// TwinCAT 3 PLC project SirupAutomat
// ProgramVersion: 3.1.0.5
// libraries:
//   Tc2_Standard, * (Beckhoff Automation GmbH)
//   Tc2_System, * (Beckhoff Automation GmbH)
//   Tc3_Interfaces, * (Beckhoff Automation GmbH)
//   Tc3_Module, * (Beckhoff Automation GmbH)
//   Tc2_OpcUa,3.3.2.0,Beckhoff Automation GmbH
//   Tc2_TcpIp,3.3.1.0,Beckhoff Automation GmbH
//   Tc2_Utilities,3.3.5.0,Beckhoff Automation GmbH
// project tree:
//   DUTs/ EKey.TcDUT, EMethod.TcDUT, EStatus.TcDUT, ECommand.TcDUT, EDosingState.TcDUT, ETimerState.TcDUT, ST_ApplicationBinaryData.TcDUT, ST_BinaryFrame.TcDUT, ST_BinaryHeader.TcDUT
//   GVLs/ DosingOuput.TcGVL, Global_Variables.TcGVL, IOStates.TcGVL, Liquids.TcGVL
//   / I_DigitalOut.TcIO, I_DosingStation.TcIO, PlcTask.TcTTO, Visualization Manager.TcVMO (not stored)
//   POUs/ FB_HardStuffDosingStation.TcPOU, FB_CO2_DosingStation.TcPOU, FB_LocalServer.TcPOU, FB_Timer.TcPOU, FB_DigitalOut.TcPOU, MAIN.TcPOU, FB_DosingStation.TcPOU
//   POUs/IP_POUs/ FB_FrameBinaryFifo.TcPOU, FB_ProtErrorFifo.TcPOU, FB_ServerApplication.TcPOU, F_ADSLOGERROR.TcPOU, F_ADSLOGHEXDATA.TcPOU, SCODE_CODE.TcPOU
//   VISUs/ HardStuff.TcVIS
// real-time tasks:
//   TASK PlcTask: cycle T#1ms, priority 20, ADS port 350
// I/O:
//   DEVICE Device 1 (EtherCAT), AmsNetId 192.168.0.103.2.1
//     Term 6 (EK1200) [EK1200-5000 EtherCAT Power supply (2A E-Bus)]
//       Term 7 (EL1008) [EL1008 8Ch. Dig. Input 24V, 3ms]
//       Term 8 (EL2008) [EL2008 8Ch. Dig. Output 24V, 0.5A]
//       Term 9 (EL2008) [EL2008 8Ch. Dig. Output 24V, 0.5A]
//       Term 10 (EL3061) [EL3061 1Ch. Ana. Input 0-10V]
//       Term 11 (EL9011) [EL9011 End Terminal]
// variable links:
//   SirupAutomat/SirupAutomat Instance <-> Device 1 (EtherCAT)/Term 6 (EK1200)/Term 10 (EL3061)
//     PlcTask Inputs/DosingOuput.iPressure <-> AI Standard/Value
//   SirupAutomat/SirupAutomat Instance <-> Device 1 (EtherCAT)/Term 6 (EK1200)/Term 7 (EL1008)
//     PlcTask Inputs/MAIN.bManualStart <-> Channel 8/Input
//     PlcTask Inputs/MAIN.fbDosingStation1.bPrefill <-> Channel 1/Input
//     PlcTask Inputs/MAIN.fbDosingStation2.bPrefill <-> Channel 2/Input
//     PlcTask Inputs/MAIN.fbDosingStation3.bPrefill <-> Channel 3/Input
//     PlcTask Inputs/MAIN.bGlassPresent <-> Channel 7/Input
//   SirupAutomat/SirupAutomat Instance <-> Device 1 (EtherCAT)/Term 6 (EK1200)/Term 8 (EL2008)
//     PlcTask Outputs/MAIN.fbDosingStation1.fbValve2.bOutput <-> Channel 2/Output
//     PlcTask Outputs/MAIN.fbDosingStation3.fbValve2.bOutput <-> Channel 6/Output
//     PlcTask Outputs/MAIN.fbDosingStation2.fbValve2.bOutput <-> Channel 4/Output
//     PlcTask Outputs/MAIN.fbDosingStation3.fbValve1.bOutput <-> Channel 5/Output
//     PlcTask Outputs/MAIN.fbDosingStation2.fbValve1.bOutput <-> Channel 3/Output
//     PlcTask Outputs/MAIN.fbDosingStation1.fbValve1.bOutput <-> Channel 1/Output
//   SirupAutomat/SirupAutomat Instance <-> Device 1 (EtherCAT)/Term 6 (EK1200)/Term 9 (EL2008)
//     PlcTask Outputs/DosingOuput.bBlowOff <-> Channel 8/Output
//     PlcTask Outputs/DosingOuput.bPump <-> Channel 7/Output

CONFIGURATION SirupAutomat
    RESOURCE PLC ON TwinCAT3
        TASK PlcTask(INTERVAL := T#1ms, PRIORITY := 20);
        PROGRAM MAIN WITH PlcTask : MAIN;
    END_RESOURCE
END_CONFIGURATION

// ---- DUTs/EKey.TcDUT
TYPE EKey :
(
	KeyCommand := 1,
	KeyVolume := 2,
	KeyStationID := 3,
	KeyStatus := 4
);
END_TYPE

// ---- DUTs/EMethod.TcDUT
TYPE EMethod :
(
	MethGet := 1,
	MethPut := 2,
	MethResponse := 3
);
END_TYPE

// ---- DUTs/EStatus.TcDUT
TYPE EStatus :
(
	NotReady,
	Ready,
	Prefilling,
	DeliverLiquid,
	Error,
	PreparingForNextDrink,
	MeasuringContent,
	RunningManualDeliver
);
END_TYPE

// ---- DUTs/ECommand.TcDUT
TYPE ECommand :
(
	None := 0,
	Deliver := 1,
	ErrorAck := 2,
	PrepareForNextDrink := 3,
	MeasureContent := 4,
	StartManualCycle
);
END_TYPE

// ---- DUTs/EDosingState.TcDUT
TYPE EDosingState :
(
	eStopped,
	eV1Opened,
    eV1AndV3Opened,
	eV1AndV2AndV3Closed,
	eV2Opened,
    eV3Opened,
	eP1Started,
	eP1Stopped,
	eV1Stopped,
	eEnd
);
END_TYPE

// ---- DUTs/ETimerState.TcDUT
TYPE ETimerState :
(
	created := 0,
	started := 1,
	outputHigh := 2,
	outputLow := 3
);
END_TYPE

// ---- DUTs/ST_ApplicationBinaryData.TcDUT
TYPE ST_ApplicationBinaryData :(* Example of binary user data structure (4 byte aligned) *)
STRUCT
	(* Adapt this structure to match your protocol needs *)
	dwMethode : DWORD;
	dwKey : DWORD;
	dwValue : DWORD;
	(* total user data size = 120 byte *)
END_STRUCT
END_TYPE

// ---- DUTs/ST_BinaryFrame.TcDUT
TYPE ST_BinaryFrame :(* Simple binary TCP/IP frame (4 byte aligned) *)
STRUCT
	head	:  ST_BinaryHeader;(* frame header *)
	data 	: ARRAY[1..PLCPRJ_BUFFER_SIZE] OF BYTE; (* user data of max. length *)
END_STRUCT
END_TYPE

// ---- DUTs/ST_BinaryHeader.TcDUT
TYPE ST_BinaryHeader :(* Simple frame header (4 byte aligned) *)
STRUCT
	dwHead		: DWORD	:= 16#BECF1234;	(* start bytes *)
	cbLength		: UDINT(0..PLCPRJ_BUFFER_SIZE) := 0;(* Max. length of attached binary data *)
	nS			: UDINT 		:= 0;		(* send counter *)
	nR			: UDINT		:= 0;		(* receive counter *)
END_STRUCT
END_TYPE

// ---- GVLs/DosingOuput.TcGVL
VAR_GLOBAL
    bPump AT %Q* : BOOL;
    bBlowOff AT %Q* : BOOL;
	iPressure AT %I* : INT;
END_VAR

// ---- GVLs/Global_Variables.TcGVL
VAR_GLOBAL CONSTANT
	PLCPRJ_MAX_CONNECTIONS						: UDINT 	:= 5;(* Max. number of server<->client connections *)
	PLCPRJ_SERVER_RESPONSE_TIMEOUT			: TIME 	:= T#10s;
	PLCPRJ_CLIENT_SEND_CYCLE_TIME				: TIME 	:= T#1s;

	PLCPRJ_RECEIVER_POLLING_CYCLE_TIME			: TIME 	:= T#200ms;
	PLCPRJ_BUFFER_SIZE							: UDINT 	:= 10000;(* Max. internal fifo/receiver buffer size *)

	(* Some project specific error codes *)
	PLCPRJ_ERROR_RECEIVE_BUFFER_OVERFLOW	: UDINT := 16#8101; (* receive fifo/buffer overflow*)
	PLCPRJ_ERROR_SEND_BUFFER_OVERFLOW		: UDINT := 16#8102;(* send fifo/buffer overflow *)
	PLCPRJ_ERROR_RESPONSE_TIMEOUT			: UDINT := 16#8103;(* receive timeout error *)
	PLCPRJ_ERROR_INVALID_FRAME_FORMAT		: UDINT := 16#8104;(* invalid frame format/data *)
END_VAR

// ---- GVLs/IOStates.TcGVL
VAR_GLOBAL
	byteInletValves AT %QB1 : BYTE;
END_VAR

// ---- GVLs/Liquids.TcGVL
VAR_GLOBAL
	Status AT %Q* : EStatus := NotReady; (*~	(OPC : 1 : available for OPC-clients)	*)
	Command AT %I* : ECommand := None; (*~	(OPC : 1 : available for OPC-clients)	*)
	StationID  AT %I* : UINT := 0; (*~	(OPC : 1 : available for OPC-clients)	*)
	Volume_ml  AT %I* : UINT := 0; (*~	(OPC : 1 : available for OPC-clients)	*)
	ErrString  AT %Q* : STRING := ''; (*~	(OPC : 1 : available for OPC-clients)	*)
	GlassPresent : BOOL := FALSE;
END_VAR

// ---- I_DigitalOut.TcIO
INTERFACE I_DigitalOut

METHOD M_On
VAR_INPUT
END_VAR
END_METHOD

 METHOD M_Off
VAR_INPUT
END_VAR
END_METHOD

END_INTERFACE

// ---- I_DosingStation.TcIO
INTERFACE I_DosingStation

METHOD M_Fill
VAR_INPUT
	tiPumpTime : TIME;
END_VAR
END_METHOD

METHOD M_Prefill
VAR_INPUT
END_VAR
END_METHOD

METHOD M_Stop
VAR_INPUT
END_VAR
END_METHOD

METHOD M_PrepareForNextDrink
VAR_INPUT
END_VAR
END_METHOD

METHOD M_GetContent_ml : BOOL
VAR_INPUT
END_VAR
END_METHOD

END_INTERFACE

// ---- POUs/MAIN.TcPOU
PROGRAM MAIN
VAR
	iStationIndex : UINT := 0;
	bGlassPresent AT %I* : BOOL;
	bManualStart AT %I* : BOOL;
	// systemState : ESystemState := eStandby;
    
	fbDosingStation1 : FB_HardStuffDosingStation;
	fbDosingStation2 : FB_HardStuffDosingStation;
    fbDosingStation3 : FB_CO2_DosingStation;
	DeliveryLiquid: INT;
	duration : TIME;
	
	A_Prefilling: INT;
	
	sLocalHost	: STRING(15) 	:= '0.0.0.0';(* Server address *)
	nLocalPort	: UDINT 		:= 200;(* Server port number *)
	bEnable		: BOOL 		:= TRUE;(* TRUE => enable server data exchange, FALSE => disable *)
	hServer		: T_HSERVER;(* Server connection handle *)
	fbApplication	: FB_ServerApplication := ( bDbg:=FALSE );(* Application (connection) instances *)

	fbCloseAll	: FB_SocketCloseAll;
	bCloseAll	: BOOL := TRUE;
	
END_VAR

A_RunIP();

CASE Status OF
	NotReady :
		IF bGlassPresent = TRUE THEN
			Status := Ready;
		ELSE
			// this works only, when no glass is present
			IF Command = MeasureContent THEN
				Status := MeasuringContent;
				iStationIndex := StationID;
				Command := None;
			END_IF
		END_IF
		
	Ready:
		IF bGlassPresent = FALSE THEN
			Status := NotReady;  
		END_IF
		
		IF Command = Deliver THEN
			Status := DeliverLiquid;
			Command := None;
		ELSIF Command = PrepareForNextDrink THEN
			Status := PreparingForNextDrink;
			Command := None;
		ELSE
			IF fbDosingStation1.bPrefill THEN 
				iStationIndex := 1;
				Status := Prefilling;
			ELSIF fbDosingStation2.bPrefill THEN
				iStationIndex := 2;
				Status := Prefilling;
			ELSIF fbDosingStation3.bPrefill THEN
				iStationIndex := 3;
				Status := Prefilling;
			ELSIF bManualStart THEN
				iStationIndex := 0;
				Status := RunningManualDeliver;
			END_IF	
		END_IF
	MeasuringContent:
		A_MeasureContent();
  
	Prefilling:
		A_Prefill();
		
	RunningManualDeliver:
		A_MixACubaLibre();
	
	DeliverLiquid:
		duration := INT_TO_TIME(UINT_TO_INT(Volume_ml) * 111);
		CASE StationID OF
			1:
				IF bGlassPresent = FALSE THEN
					fbDosingStation1.M_Stop();
					Status := Error;
				ELSE
					fbDosingStation1.M_Fill(duration);
					IF fbDosingStation1.bFinished THEN
						Status := NotReady;
					END_IF
				END_IF
		
			2:
				IF bGlassPresent = FALSE THEN
					fbDosingStation2.M_Stop();
					Status := Error;
				ELSE
					fbDosingStation2.M_Fill(duration);
					IF fbDosingStation2.bFinished THEN
						Status := NotReady;
					END_IF
				END_IF
				
			3:
				IF bGlassPresent = FALSE THEN
					fbDosingStation3.M_Stop();
					Status := Error;
				ELSE
					fbDosingStation3.M_Fill(duration);
					IF fbDosingStation3.bFinished THEN
						Status := NotReady;
					END_IF
				END_IF		
	
		END_CASE

	Error:
		IF Command = ErrorAck THEN
			Status := NotReady;
		END_IF
		
	PreparingForNextDrink:
		CASE StationID OF
			1:
				IF bGlassPresent = FALSE THEN
					fbDosingStation1.M_Stop();
					Status := Error;
				ELSE
					fbDosingStation1.M_PrepareForNextDrink();
					IF fbDosingStation1.bFinished THEN
						Status := NotReady;
					END_IF
				END_IF
		
			2:
				IF bGlassPresent = FALSE THEN
					fbDosingStation2.M_Stop();
					Status := Error;
				ELSE
					fbDosingStation2.M_PrepareForNextDrink();
					IF fbDosingStation2.bFinished THEN
						Status := NotReady;
					END_IF
				END_IF
				
			3:
				IF bGlassPresent = FALSE THEN
					fbDosingStation3.M_Stop();
					Status := Error;
				ELSE
					fbDosingStation3.M_PrepareForNextDrink();
					IF fbDosingStation3.bFinished THEN
						Status := NotReady;
					END_IF
				END_IF		
	
		END_CASE		
		
END_CASE

ACTION A_Prefill:
IF iStationIndex = 1 THEN
    fbDosingStation1.M_Prefill();
    IF fbDosingStation1.bFinished THEN
		iStationIndex := 0;
		Status := NotReady;
    END_IF
ELSIF  iStationIndex = 2  THEN
    fbDosingStation2.M_Prefill();
    IF fbDosingStation2.bFinished THEN
		iStationIndex := 0;
		Status := NotReady;
    END_IF
ELSIF  iStationIndex = 3  THEN
    fbDosingStation3.M_Prefill();
    IF fbDosingStation3.bFinished THEN
		iStationIndex := 0;
		Status := NotReady;
    END_IF
END_IF
END_ACTION

ACTION A_RunIP:
IF bCloseAll THEN(*On PLC reset or program download close all old (opened) connections *)
	bCloseAll := FALSE;

	(* Initialize server handle *)
	F_CreateServerHnd( 	sSrvNetID 	:= '',
						sLocalHost 	:= sLocalHost,
						nLocalPort	:= nLocalPort,
						nMode 		:= CONNECT_MODE_ENABLEDBG,(* Enable debug messages *)
						bEnable 		:= FALSE,(* TRUE = leave listener socket open, FALSE = close listener socket after last connection ist closed too *)
						hServer 		:= hServer );


	fbCloseAll( bExecute:= TRUE );
ELSE
	fbCloseAll( bExecute:= FALSE );
END_IF


IF NOT fbCloseAll.bBusy THEN
	(* trigger the execution of every connection instance *)
	fbApplication( hServer := hServer, bEnable := bEnable );
END_IF
END_ACTION

ACTION A_MeasureContent:
IF iStationIndex = 1 THEN
    fbDosingStation1.M_GetContent_ml();
    IF fbDosingStation1.bFinished THEN
		iStationIndex := 0;
		Status := NotReady;
    END_IF
ELSIF  iStationIndex = 2  THEN
    fbDosingStation2.M_GetContent_ml();
    IF fbDosingStation2.bFinished THEN
		iStationIndex := 0;
		Status := NotReady;
    END_IF
ELSIF  iStationIndex = 3  THEN
    fbDosingStation3.M_GetContent_ml();
    IF fbDosingStation3.bFinished THEN
		iStationIndex := 0;
		Status := NotReady;
    END_IF
END_IF
END_ACTION

ACTION A_MixACubaLibre:
IF iStationIndex = 0 THEN
    iStationIndex := 3;
END_IF

IF iStationIndex = 1 THEN
    // the Rum
	fbDosingStation1.M_Fill(INT_TO_TIME(UINT_TO_INT(10) * 111));
    IF fbDosingStation1.bFinished THEN
        iStationIndex := 4;
    END_IF
END_IF

IF iStationIndex = 2 THEN
    // the Vodka is not used yet 
	fbDosingStation2.M_Fill(TIME#16S);
    IF fbDosingStation2.bFinished THEN
        iStationIndex := 3;
    END_IF
END_IF

IF iStationIndex = 3 THEN
    // the CocaCola 
	fbDosingStation3.M_Fill(INT_TO_TIME(UINT_TO_INT(200) * 111));
    IF fbDosingStation3.bFinished THEN
        iStationIndex := 1;
    END_IF
END_IF

IF iStationIndex = 4 THEN
    iStationIndex := 0;
	Status := NotReady;
END_IF
END_ACTION

END_PROGRAM

// ---- POUs/FB_HardStuffDosingStation.TcPOU
FUNCTION_BLOCK FB_HardStuffDosingStation EXTENDS FB_DosingStation
VAR_INPUT
	bPrefill AT %I* : BOOL;
END_VAR
VAR_OUTPUT
	bFinished : BOOL := TRUE;
	error : BOOL := FALSE;
END_VAR
VAR
	fbT1 : FB_Timer;
	dosingState : EDosingState := eStopped;
	fbValve1 : FB_DigitalOut;
	fbValve2 : FB_DigitalOut;
	
	iStartPressure : INT;
	iActualPressure : INT;
	iDeltaPressure : INT;
	iContentMeasurementTimeout : TIME := TIME#5S;
END_VAR
VAR_EXTERNAL
    bPump : BOOL;
END_VAR

;

METHOD M_Fill
VAR_INPUT
	    tiPumpTime : TIME := TIME#2S;
END_VAR

CASE dosingState OF
	eStopped :
		// wait for start
   		bFinished := FALSE;
        fbValve2.M_On();
        dosingState := eV2Opened;
	eV2Opened :
		fbT1.M_Start(TIME#1S);
		IF fbT1.bTimeout THEN
			fbValve1.M_On();
			dosingState := eV1Opened;
		END_IF
	eV1Opened :
		fbT1.M_Start(TIME#1S);
		IF fbT1.bTimeout THEN
			bPump := TRUE;
			dosingState := eP1Started;
		END_IF
	eP1Started :
		fbT1.M_Start(tiPumpTime);
		IF fbT1.bTimeout THEN
			bPump := FALSE;
			dosingState := eP1Stopped;
		END_IF
	eP1Stopped :
		fbT1.M_Start(TIME#1S);
		IF fbT1.bTimeout THEN
			fbValve1.M_Off();
			dosingState := eV1Stopped;
		END_IF
	eV1Stopped :
		fbT1.M_Start(TIME#10S);
		IF fbT1.bTimeout THEN
			fbValve2.M_Off();
			dosingState := eEnd;
		END_IF
	eEnd :
   		bFinished := TRUE;
		dosingState := eStopped;
END_CASE
END_METHOD

METHOD M_Prefill
VAR_INPUT
END_VAR
CASE dosingState OF
	eStopped :
		// wait for start
   		bFinished := FALSE;
        fbValve2.M_On();
        dosingState := eV2Opened;
	eV2Opened :
		fbT1.M_Start(TIME#0S);
		IF fbT1.bTimeout THEN
			fbValve1.M_On();
			dosingState := eV1Opened;
		END_IF
	eV1Opened :
		fbT1.M_Start(TIME#0S);
		IF fbT1.bTimeout THEN
			bPump := TRUE;
			dosingState := eP1Started;
		END_IF
	eP1Started :
		IF NOT bPrefill THEN
			bPump := FALSE;
			dosingState := eP1Stopped;
		END_IF
	eP1Stopped :
		fbT1.M_Start(TIME#1S);
		IF fbT1.bTimeout THEN
			fbValve1.M_Off();
			dosingState := eV1Stopped;
		END_IF
	eV1Stopped :
		fbT1.M_Start(TIME#5S);
		IF fbT1.bTimeout THEN
			fbValve2.M_Off();
			dosingState := eEnd;
		END_IF
	eEnd :
   		bFinished := TRUE;
		dosingState := eStopped;
END_CASE
END_METHOD

METHOD M_Stop
VAR_INPUT
END_VAR
fbValve2.M_Off();
fbValve1.M_Off();
bPump := FALSE;	
dosingState := eStopped;
bFinished := TRUE;
END_METHOD

METHOD M_PrepareForNextDrink
VAR_INPUT
END_VAR
CASE dosingState OF
	eStopped :
		// wait for start
		bFinished := FALSE;
        fbValve2.M_On();
        dosingState := eV2Opened;
	eV2Opened :
		fbT1.M_Start(TIME#10S);
		IF fbT1.bTimeout THEN
			fbValve2.M_Off();
			dosingState := eEnd;
		END_IF
	eEnd :
   		bFinished := TRUE;
		dosingState := eStopped;		
END_CASE
END_METHOD

METHOD M_GetContent_ml : BOOL
VAR_INPUT
END_VAR
VAR
END_VAR
CASE dosingState OF
	eStopped :
		// wait for start
   		bFinished := FALSE;
        // open the 2 valves (the blow off valve is valve 3) to release overpressure of the CO2 bottle
        bBlowOff := TRUE;
        fbValve1.M_On();
        dosingState := eV1AndV3Opened;
    eV1AndV3Opened :    
		fbT1.M_Start(TIME#2S);
		IF fbT1.bTimeout THEN
            // after a timeout close the blow off valve and the inlet
			bBlowOff := FALSE;
			fbValve1.M_Off();
			iStartPressure := iPressure;
			bPump := TRUE;
			dosingState := eV1AndV2AndV3Closed;
		END_IF
	eV1AndV2AndV3Closed :
		// now everything is closed, pump it up
		fbT1.M_Start(iContentMeasurementTimeout);
		IF fbT1.bTimeout THEN
			iActualPressure := iPressure;
			bPump := FALSE;
			// let the pressure escape
			bBlowOff := TRUE;
			dosingState := eV3Opened;
		END_IF
	eV3Opened :
		fbT1.M_Start(TIME#1S);
		IF fbT1.bTimeout THEN
			iDeltaPressure := iActualPressure - iStartPressure;
			bBlowOff := FALSE;
			dosingState := eEnd;
		END_IF
	eEnd :
   		bFinished := TRUE;
		dosingState := eStopped;
END_CASE
END_METHOD

END_FUNCTION_BLOCK

// ---- POUs/FB_DosingStation.TcPOU
FUNCTION_BLOCK FB_DosingStation IMPLEMENTS I_DosingStation
VAR_INPUT
END_VAR
VAR_OUTPUT
END_VAR
VAR
END_VAR

METHOD M_Fill
VAR_INPUT
	tiPumpTime : TIME;
END_VAR
END_METHOD

METHOD M_Prefill
VAR_INPUT
END_VAR
END_METHOD

METHOD M_Stop
VAR_INPUT
END_VAR
END_METHOD

METHOD M_PrepareForNextDrink
VAR_INPUT
END_VAR
END_METHOD

METHOD M_GetContent_ml : BOOL
VAR_INPUT
END_VAR
;
END_METHOD

END_FUNCTION_BLOCK

// ---- POUs/FB_Timer.TcPOU
FUNCTION_BLOCK FB_Timer
VAR_INPUT
	tiTimeout : TIME;
END_VAR
VAR_OUTPUT
	bTimeout : BOOL;
	iIndex : UINT := 0;
	toggler : BOOL := FALSE;
END_VAR
VAR
	timer : TON;
	toggleTimer : TON;
	countUpTimer : TON;
	elapsed : TIME;
	state : ETimerState := created;
END_VAR

;

METHOD M_ToggleOutput
VAR_INPUT
END_VAR
elapsed := toggleTimer.ET;
CASE state OF 
	created :
		//onTimer.PT := TIME#4S;
		toggleTimer(IN := TRUE, PT := TIME#4S);
		state := outputLow;
	outputLow :
		IF NOT toggleTimer.Q THEN
			toggleTimer(IN := TRUE, PT := TIME#1S);
		END_IF
		IF toggleTimer.Q THEN
			toggleTimer(IN := FALSE);
			state := outputHigh;
			toggler := TRUE;
		END_IF
	outputHigh :		
		IF NOT toggleTimer.Q THEN
			toggleTimer(IN := TRUE, PT := TIME#1S);
		END_IF
		IF toggleTimer.Q THEN
			toggleTimer(IN := FALSE);
			state := outputLow;
			toggler := FALSE;
		END_IF
END_CASE
END_METHOD

METHOD M_CountUp
VAR_INPUT
END_VAR
IF NOT countUpTimer.Q THEN
	countUpTimer( IN := TRUE, PT := TIME#2S );
END_IF

IF countUpTimer.Q THEN
	countUpTimer( IN := FALSE ); 
	iIndex := iIndex + 1;
END_IF
END_METHOD

METHOD M_Start
VAR_INPUT
	tiTimeout : TIME;
END_VAR
IF NOT timer.Q THEN
	bTimeout := FALSE; 
	timer( IN := TRUE, PT := tiTimeout );
END_IF

IF timer.Q THEN
	timer( IN := FALSE );
	bTimeout := TRUE; 
END_IF
timer();
END_METHOD

END_FUNCTION_BLOCK

// ---- POUs/FB_DigitalOut.TcPOU
FUNCTION_BLOCK FB_DigitalOut IMPLEMENTS I_DigitalOut
VAR_INPUT
END_VAR
VAR_OUTPUT
	bOutput AT %Q* : BOOL := FALSE;
END_VAR
VAR
END_VAR

METHOD M_Off
bOutput := FALSE;
END_METHOD

METHOD M_On
bOutput := TRUE;
END_METHOD

END_FUNCTION_BLOCK

// ---- POUs/FB_CO2_DosingStation.TcPOU
FUNCTION_BLOCK FB_CO2_DosingStation  IMPLEMENTS I_DosingStation
VAR_INPUT
	bPrefill AT %I* : BOOL;
END_VAR
VAR_OUTPUT
	bFinished : BOOL := TRUE;
END_VAR
VAR
	fbT1 : FB_Timer;
	dosingState : EDosingState := eStopped;
	fbValve1 : FB_DigitalOut;
	fbValve2 : FB_DigitalOut;
END_VAR
VAR_EXTERNAL
    // the global enable/disable for the pump and the blow off valve
    bPump : BOOL;
    bBlowOff : BOOL;
END_VAR

;

METHOD M_Fill
VAR_INPUT
    tiPumpTime : TIME := TIME#2S;
END_VAR
CASE dosingState OF
	eStopped :
		// wait for start
   		bFinished := FALSE;
        // open the 2 valves (the blow off valve is valve 3) to release overpressure of the CO2 bottle
        bBlowOff := TRUE;
        fbValve1.M_On();
        dosingState := eV1AndV3Opened;
    eV1AndV3Opened :    
		fbT1.M_Start(TIME#2S);
		IF fbT1.bTimeout THEN
            // after a timeout close the blow off valve and open the outlet
			bBlowOff := FALSE;
			fbValve2.M_On();
			dosingState := eV2Opened;
		END_IF
	eV2Opened :
		fbT1.M_Start(TIME#1S);
		IF fbT1.bTimeout THEN
			fbValve1.M_On();
			dosingState := eV1Opened;
		END_IF
	eV1Opened :
		fbT1.M_Start(TIME#1S);
		IF fbT1.bTimeout THEN
			bPump := TRUE;
			dosingState := eP1Started;
		END_IF
	eP1Started :
		fbT1.M_Start(tiPumpTime);
		IF fbT1.bTimeout THEN
			bPump := FALSE;
			dosingState := eP1Stopped;
		END_IF
	eP1Stopped :
		fbT1.M_Start(TIME#1S);
		IF fbT1.bTimeout THEN
			fbValve1.M_Off();
			dosingState := eV1Stopped;
		END_IF
	eV1Stopped :
		fbT1.M_Start(TIME#10S);
		IF fbT1.bTimeout THEN
			fbValve2.M_Off();
			dosingState := eEnd;
		END_IF
	eEnd :
   		bFinished := TRUE;
		dosingState := eStopped;
END_CASE
END_METHOD

METHOD M_Prefill
VAR_INPUT
END_VAR
CASE dosingState OF
	eStopped :
		// wait for start
		bFinished := FALSE;
		// open the 2 valves (the blow-off valve an inlet of the bottle) to release overpressure of the CO2 bottle
		bBlowOff := TRUE;
		fbValve1.M_On();
		dosingState := eV1AndV3Opened;
	eV1AndV3Opened :
        // let the CO2 blow-off for a short time    
		fbT1.M_Start(TIME#2S);
		IF fbT1.bTimeout THEN
			// after a timeout close the blow-off valve and open the outlet
            // let the inlet open
			bBlowOff := FALSE;
			fbValve2.M_On();
            // jump directly to the pump, because the inlet ist already open
			dosingState := eV1Opened;
		END_IF
	eV2Opened :
        // don't wait 
		fbT1.M_Start(TIME#0S);
		IF fbT1.bTimeout THEN
			fbValve1.M_On();
			dosingState := eV1Opened;
		END_IF
	eV1Opened :
        // don't wait 
		fbT1.M_Start(TIME#0S);
		IF fbT1.bTimeout THEN
			bPump := TRUE;
			dosingState := eP1Started;
		END_IF
	eP1Started :
		IF NOT bPrefill THEN
			bPump := FALSE;
			dosingState := eP1Stopped;
		END_IF
	eP1Stopped :
        // don't wait the Coca Cola pooring out
        // therefore close inlet and outlet simultaneously
		fbT1.M_Start(TIME#0S);
		IF fbT1.bTimeout THEN
			fbValve1.M_Off();
			fbValve2.M_Off();
			dosingState := eEnd;
		END_IF
	eV1Stopped :
		fbT1.M_Start(TIME#5S);
		IF fbT1.bTimeout THEN
			fbValve2.M_Off();
			dosingState := eEnd;
		END_IF
	eEnd :
		bFinished := TRUE;
		dosingState := eStopped;
END_CASE
END_METHOD

METHOD M_Stop
VAR_INPUT
END_VAR
fbValve2.M_Off();
fbValve1.M_Off();
bPump := FALSE;	
dosingState := eStopped;
bFinished := TRUE;
END_METHOD

METHOD M_PrepareForNextDrink
VAR_INPUT
END_VAR
bFinished := TRUE;
dosingState := eStopped;
END_METHOD

METHOD M_GetContent_ml : BOOL
VAR_INPUT
END_VAR
VAR
	uiStartPressure : UINT;
	uiActualPressure : UINT;
END_VAR
;
END_METHOD

END_FUNCTION_BLOCK

// ---- POUs/IP_POUs/FB_ServerApplication.TcPOU
FUNCTION_BLOCK FB_ServerApplication
(* Sample server application. Adapt this code to match your needs. *)
VAR_IN_OUT
	hServer 	: T_HSERVER;(* Server connection handle *)
END_VAR
VAR_INPUT
	bDbg		: BOOL 	:= FALSE;(* TRUE => Enable debug output, FALSE => Disable *)
	bEnable		: BOOL 	:= TRUE;(* TRUE => Enable connection, FALSE => Disable *)
END_VAR
VAR_OUTPUT
	eState		: E_SocketConnectionState := eSOCKET_DISCONNECTED;(* TCP/IP connection state *)
END_VAR
VAR
	bCaseError : BOOL;
	fromClient	: ST_ApplicationBinaryData; (* Rx user data *)
	toClient	: ST_ApplicationBinaryData; (* Tx user data *)

	fbServer		: FB_LocalServer;(* Implements one server->client connection *)
	tx 			: FB_FrameBinaryFifo; (* Tx fifo *)
	rx 			: FB_FrameBinaryFifo; (* Rx fifo *)
	errors		: FB_ProtErrorFifo; (* Error fifo *)
END_VAR

(* ------------------------------------- trigger data exchange ----------------------------------------------------------------------------------------------*)
fbServer( bDbg := bDbg, hServer := hServer, rx := rx, tx := tx, errors := errors, bEnable := bEnable, eState => eState  );



(*----------------------------------------------- fetch rx data and send them back to the client ---------------------------------------------------------------------------------------------------- *)
IF eState = eSOCKET_CONNECTED THEN

	REPEAT
		rx.A_RemoveHead( pGet := ADR( fromClient ), cbGet := SIZEOF( fromClient ) );(* fetch data from rx fifo *)
		IF rx.bOk THEN(* success *)

			IF fromClient.dwMethode = MethPut THEN
				CASE fromClient.dwKey OF
					KeyCommand:
						Command  := DWORD_TO_INT(fromClient.dwValue);
						bCaseError := FALSE;
					KeyVolume:
						Volume_ml := DWORD_TO_INT(fromClient.dwValue);
						bCaseError := FALSE;
					KeyStationID:
					    StationID := DWORD_TO_INT(fromClient.dwValue);
						bCaseError := FALSE;
				ELSE
					bCaseError := TRUE;
				END_CASE
				// don't leave him with no response
				toClient.dwMethode := MethResponse;
				toClient.dwKey := fromClient.dwKey;
				toClient.dwValue := fromClient.dwValue;
			ELSIF  fromClient.dwMethode = MethGet THEN
				CASE fromClient.dwKey OF
					KeyStatus:
						toClient.dwMethode := MethResponse;
						toClient.dwKey := KeyStatus;
						toClient.dwValue := Status;
						bCaseError := FALSE;
				ELSE
					bCaseError := TRUE;
				END_CASE
			END_IF
		
			(* send data back to the client *)
			tx.A_AddTail( pPut := ADR(  toClient ), cbPut := SIZEOF( toClient ) );(* put user data to the tx fifo *)
			IF NOT tx.bOk THEN(* fifo overflow: log error *)
				errors.A_AddTail( putError := PLCPRJ_ERROR_SEND_BUFFER_OVERFLOW );
			END_IF

		END_IF
	UNTIL NOT rx.bOk
	END_REPEAT

END_IF

(*-------------------------------------- get error messages from error fifo ----------------------------------------------------------------------------- *)
REPEAT
	errors.A_RemoveHead( bDbg := bDbg );
	IF errors.bOk THEN
		;(* TODO: Implement error handler *)
	END_IF
UNTIL NOT errors.bOk
END_REPEAT

END_FUNCTION_BLOCK

// ---- POUs/FB_LocalServer.TcPOU
FUNCTION_BLOCK FB_LocalServer
(* 	This function block implements simple TCP/IP server protocol.
	The max. size of binary tx/rx data has to be <= PLCPRJ_BUFFER_SIZE  *)
VAR_IN_OUT
	hServer		: T_HSERVER;(* Server connection handle *)
	tx			: FB_FrameBinaryFifo;(* TX fifo *)
	rx			: FB_FrameBinaryFifo;(* RX fifo *)
	errors 		: FB_ProtErrorFifo;(* Error message fifo *)
END_VAR
VAR_INPUT
	bDbg		: BOOL := FALSE; (* TRUE => Enable debug output, FALSE => Disable debug output *)
	bEnable		: BOOL := TRUE;(* TRUE => Enable/connect, FALSE => Disable/disconnect *)
END_VAR
VAR_OUTPUT
	eState		: E_SocketConnectionState := eSOCKET_DISCONNECTED;(* TCP/IP connection state *)
END_VAR
VAR
	fbConnect	: FB_ServerClientConnection;(* create/release TCP/IP connection *)
	fbSend		: FB_SocketSend;(* send TCP/IP data *)
	fbReceive	: FB_SocketReceive;(* receive TCP/IP data *)
	state 		: BYTE;(* global state *)
	tx_state 	: BYTE;(* tx state *)
	rx_state 	: BYTE;(* rx state *)

	nS			: UDINT;(* Send frame counter *)
	nR			: UDINT;(* Received frame counter *)

	txFrame		: ST_BinaryFrame;(* Tx frame buffer (inclusive header) *)
	rxFrame		: ST_BinaryFrame;(* Rx frame buffer (inclusive header) *)
	cbReceived	: UDINT;(* Count of received data bytes *)
	cbRx		: UDINT;(* Rx frame byte size *)

	bDisconnect	: BOOL;(* Disconnect flag, if set the socket will be closed *)
	pollTimer	: TON;(* Rx data poll timer *)
	bAbort		: BOOL;(* Flag to abort frame parsing loop *)
	sID			: STRING(20) := '';
END_VAR

CASE state OF
	0:(* init state *)
		rx.A_Reset( bDbg := bDbg );(* Reset RX fifo (optional) *)
		tx.A_Reset( bDbg := bDbg );(* Reset TX fifo (optional) *)
		errors.A_Reset( bDbg := bDbg );(* Reset error fifo (optional) *)

		pollTimer( IN := FALSE, PT := PLCPRJ_RECEIVER_POLLING_CYCLE_TIME );
		bDisconnect 	:= FALSE;(* Reset disconnect flag *)
		cbReceived 	:= 0;(* Reset number of received data bytes *)
		nR 			:= 0;(* Reset receive frame counter *)
		nS 			:= 0;(* Reset send frame counter *)
		tx_state 		:= 0;(* Reset tx state machine *)
		rx_state 		:= 0;(* Reset rx state machine *)
		state 		:= 1;(* Go to the next step *)

	1:(* connect *)
		fbConnect( 	eMode		:= eACCEPT_ALL,
					bEnable		:= bEnable,
					tReconnect	:= T#1s,
					hServer		:= hServer,
					eState		=> eState );
		IF NOT fbConnect.bBusy THEN

			(* Create identification string used by debug messages *)
			sID 			:= CONCAT( CONCAT('[', DWORD_TO_HEXSTR(fbConnect.hSocket.handle, 4, FALSE) ), ']' );
			tx.sDesc		:= CONCAT( 'SRV.Tx', sID );
			rx.sDesc		:= CONCAT( 'SRV.Rx', sID );
			errors.sDesc 	:= CONCAT( 'SRV.Err', sID );

			IF NOT fbConnect.bError THEN
				IF eState = eSOCKET_CONNECTED THEN
					state 		:= 2;
				END_IF
			ELSE(* error => log error *)
				errors.A_AddTail( putError := fbConnect.nErrID );
			END_IF
		END_IF

	2:(* data exchange state *)
		bDisconnect := NOT bEnable OR bDisconnect;(* user/internal disconnect requested? *)
		IF bDisconnect AND (tx_state = 0) AND (rx_state = 0) THEN
			state := 3;(* disconnect *)
		ELSE

			(* get rx data *)
			CASE rx_state OF
				0:
					IF NOT bDisconnect THEN
						pollTimer( IN := TRUE );
						IF pollTimer.Q THEN
							IF rx.cbFree >= SIZEOF(rxFrame.data) THEN(* check free rx fifo space *)
								pollTimer( IN := FALSE );

								fbReceive( bExecute := FALSE );
								fbReceive( 	sSrvNetId	:= '',
											hSocket		:= fbConnect.hSocket,
											cbLen		:= SIZEOF(rxFrame) - cbReceived,
											pDest		:= ADR(rxFrame) + cbReceived,
											bExecute	:= TRUE,
											tTimeout		:= T#5s );
								rx_state := 1;
							END_IF
						END_IF
					END_IF
				1:(* wait until receive not busy *)
					fbReceive( bExecute := FALSE );
					IF NOT fbReceive.bBusy THEN
						rx_state := 0;
						IF NOT fbReceive.bError THEN
							IF fbReceive.nRecBytes > 0 THEN (* some bytes received *)

								pollTimer( PT := T#0s );(* increase polling speed *)
								cbReceived := cbReceived + fbReceive.nRecBytes;

								(* parse received bytes *)
								REPEAT
									bAbort := TRUE;(* set flag *)
									IF cbReceived >= SIZEOF(rxFrame.head) THEN (* all header bytes received => check header data *)

										IF (rxFrame.head.dwHead = 16#BECF1234) (* check start bytes *)
										AND (rxFrame.head.nS = nR )(* check counter (send counter == expected receive counter?) *)
										AND (rxFrame.head.cbLength <= SIZEOF( rxFrame.data))(* check frame (user data) length *)
										THEN

											cbRx := SIZEOF(rxFrame.head) + rxFrame.head.cbLength;(* calculate the length of the rx frame *)
											IF cbReceived >= cbRx  THEN (* all frame bytes received? *)

												rx.A_AddTail( bDbg := bDbg, pPut := ADR( rxFrame.data ), cbPut := rxFrame.head.cbLength );(* add user data to the rx fifo *)
												IF rx.bOk THEN
													nR := nR + 1;(* increment receive counter *)

													MEMMOVE( ADR( rxFrame ), ADR( rxFrame ) + cbRx,  cbReceived - cbRx );(* shift the remaining rx bytes *)
													cbReceived := cbReceived - cbRx;(* recalculate the size of the remaining rx bytes *)

													IF rx.cbFree >= SIZEOF(rxFrame.data) THEN
														bAbort := FALSE;(* reset flag, try to parse next frame *)
													END_IF
												ELSE (* fifo overflow => log error and disconnect *)
													errors.A_AddTail( putError := PLCPRJ_ERROR_RECEIVE_BUFFER_OVERFLOW );
													bDisconnect := TRUE;(* set flag *)
												END_IF

(*											ELSE repeat reading *)
											END_IF

										ELSE(* receive error: invalid frame format/data *)
											errors.A_AddTail( putError := PLCPRJ_ERROR_INVALID_FRAME_FORMAT );
											bDisconnect := TRUE;(* set flag *)
										END_IF
(*									ELSE repeat reading *)
									END_IF (* IF cbReceived >= SIZEOF(rxFrame.head) THEN *)

								UNTIL bAbort
								END_REPEAT

							ELSE(* fbReceive.nRecBytes = 0, repeat reading *)
								pollTimer( PT := PLCPRJ_RECEIVER_POLLING_CYCLE_TIME );(* slow down the polling cycle *)
							END_IF(* IF fbReceive.nRecBytes > 0 THEN *)
						ELSE(* receive error => log error and disconnect *)
							errors.A_AddTail( putError := fbReceive.nErrId );
							bDisconnect := TRUE;(* set flag *)
						END_IF

					END_IF(*IF NOT fbReceive.bBusy THEN*)

			END_CASE


			(* send tx data *)
			CASE tx_state OF
				0:
					IF NOT bDisconnect THEN
						tx.A_RemoveHead( bDbg := bDbg, pGet := ADR( txFrame.data ), cbGet := SIZEOF( txFrame.data ) );(* remove oldest user data entry *)
						IF tx.bOk THEN(* success *)

							(* append/create some protocol header  *)
							txFrame.head.dwHead 	:= 16#BECF1234;(* frame start bytes *)
							txFrame.head.cbLength := tx.cbReturn;(* set length of user data *)
							txFrame.head.nS 		:= nS;(* number of send frames *)
							txFrame.head.nR 		:= nR;(* number of received frames *)

							(* send frame *)
							fbSend( bExecute := FALSE );
							fbSend(	sSrvNetID 	:= '',
									hSocket		:= fbConnect.hSocket,
									cbLen		:= SIZEOF(txFrame.head) + txFrame.head.cbLength,(* size of header + size of user data *)
									pSrc		:= ADR(txFrame),(* pointer to the frame data *)
									bExecute	:= TRUE,
									tTimeout 		:= T#5s );

							tx_state := 1;
						END_IF
					END_IF
				1:(* wait until send not busy *)
					fbSend( bExecute := FALSE );
					IF NOT fbSend.bBusy THEN
						tx_state := 0;
						IF NOT fbSend.bError THEN(* no error *)
							nS := nS + 1;(* increment the number of send frames *)
						ELSE(* send error => log error and disconnect *)
							errors.A_AddTail( putError := fbSend.nErrId );
							bDisconnect := TRUE;(* set flag *)
						END_IF
					END_IF
			END_CASE


		END_IF


	3:(* disconnect *)
		fbConnect( hServer := hServer, bEnable:= FALSE, eState=>eState );
		IF eState = eSOCKET_DISCONNECTED THEN
			state := 0;
		END_IF


END_CASE

END_FUNCTION_BLOCK

// ---- POUs/IP_POUs/FB_FrameBinaryFifo.TcPOU
FUNCTION_BLOCK FB_FrameBinaryFifo
(* Tx/Rx (binary data) fifo control function block *)
VAR_INPUT
	sDesc		: STRING(20)	:= 'Unknown';(* Debug message description string (allows the identification of log message source) *)
	bDbg		: BOOL 		:= FALSE; (* TRUE => Enable debug output, FALSE => Disable *)
	pPut			: DWORD 	:= 0;(* Address/pointer to the source data  *)
	cbPut		: UDINT(0..PLCPRJ_BUFFER_SIZE) := 0;(* Byte size of the source data *)
	pGet		: DWORD 	:= 0;(* Address/pointer to the destination buffer *)
	cbGet		: UDINT(0..PLCPRJ_BUFFER_SIZE) := 0;(* Max. byte size of the destination buffer *)
END_VAR
VAR_OUTPUT
	bOk			: BOOL; 	 (* TRUE = New entry added or removed succesfully, FALSE = Fifo overflow or fifo empty *)
	cbReturn		: UDINT 	:= 0; (* Number of get/removed data bytes *)
	nCount		: UDINT	:= 0;	(* Number of fifo entries *)
	cbFree		: UDINT	:= 0;	(* Free buffer space *)
END_VAR
VAR
	buffer		: ARRAY[-3..PLCPRJ_BUFFER_SIZE] OF BYTE;(* Internal buffer memory *)
	fbBuffer 		: FB_MemRingBuffer;(* Basic (lower level) buffer control function block *)
END_VAR

;

ACTION A_AddTail:
(* adds new fifo entry *)
fbBuffer.A_AddTail(  	pWrite := pPut, cbWrite := cbPut,
					pBuffer:= ADR(buffer), cbBuffer:= SIZEOF(buffer),
					bOk=>bOk, nCount=>nCount );
IF bOk THEN
	cbFree := PLCPRJ_BUFFER_SIZE - fbBuffer.cbSize;(* calculate the free buffer space *)
	IF bDbg THEN(* log message *)
		F_ADSLOGHEXDATA( CONCAT( sDesc, '<=' ), pPut, cbPut );
	END_IF
END_IF
END_ACTION

ACTION A_RemoveHead:
(* removes oldest fifo entry *)
fbBuffer.A_RemoveHead( 	pRead := pGet, cbRead := cbGet,
						pBuffer:= ADR(buffer), cbBuffer:= SIZEOF(buffer),
						bOk=>bOk, nCount=>nCount, cbReturn=>cbReturn );
IF bOk THEN
	cbFree := PLCPRJ_BUFFER_SIZE - fbBuffer.cbSize;(* calculate the free buffer space *)
	IF bDbg THEN(* log message *)
		F_ADSLOGHEXDATA( CONCAT( sDesc, '=>' ), pGet, cbReturn );
	END_IF
END_IF
END_ACTION

ACTION A_Reset:
(* resets fifo = clears all data *)
fbBuffer.A_Reset( 	pBuffer:= ADR(buffer), cbBuffer:= SIZEOF(buffer),
				bOk=>bOk, nCount=>nCount, cbReturn =>cbReturn );

cbFree := PLCPRJ_BUFFER_SIZE;
END_ACTION

END_FUNCTION_BLOCK

// ---- POUs/IP_POUs/F_ADSLOGHEXDATA.TcPOU
FUNCTION F_ADSLOGHEXDATA : DINT
(* This function logs hexadecimal data to the TwinCAT System Log View *)
VAR_INPUT
	sPrefix		: STRING(20);(* Debug message prefix string (allows the identification of log message source) *)
	pBuffer		: DWORD;(* Address of source buffer *)
	cbBuffer		: UDINT;(* Byte size of source buffer *)
END_VAR
VAR
	fbSplit	: FB_MemBufferSplit;
	sArg	: T_MaxString;
	sFormat 	: STRING;
END_VAR

IF pBuffer = 0 OR cbBuffer = 0 THEN
	RETURN;
END_IF

sFormat := CONCAT( sPrefix, '%s' );
fbSplit.eCmd := eEnumCmd_First;

REPEAT
	fbSplit( pBuffer := pBuffer, cbBuffer := cbBuffer, cbSize := 32 );(* split binary data to 64 byte segments *)
	IF fbSplit.bOk THEN

		sArg := DATA_TO_HEXSTR( pData := fbSplit.pSegment, cbData := fbSplit.cbSegment, FALSE );(* convert binary data to hex string *)

		F_ADSLOGHEXDATA := ADSLOGSTR( ADSLOG_MSGTYPE_HINT OR ADSLOG_MSGTYPE_LOG, sFormat, sArg );(* log hex string *)

		sFormat := '%s';
		fbSplit.eCmd := eEnumCmd_Next;
	END_IF
UNTIL NOT fbSplit.bOk
END_REPEAT

END_FUNCTION

// ---- POUs/IP_POUs/FB_ProtErrorFifo.TcPOU
FUNCTION_BLOCK FB_ProtErrorFifo
(* Protocol error fifo control function block *)
VAR_INPUT
	sDesc		: STRING(20)	:= 'Unknown';(* Debug message description string (allows the identification of message source) *)
	bDbg		: BOOL 		:= FALSE; (* TRUE => Enable debug output, FALSE => Disable *)
	putError	: UDINT 		:= 0; (* Error code to add (write) to the fifo *)
END_VAR
VAR_OUTPUT
	bOk			: BOOL; 	 	(* TRUE = New entry added or removed succesfully, FALSE = Fifo overflow or fifo empty *)
	getError	: UDINT		:= 0; (* Error code get/removed (read) from fifo *)
	nCount		: UDINT		:= 0;	(* Number of fifo entries *)
END_VAR
VAR
	buffer		: ARRAY[-3..20] OF BYTE;(* Internal buffer memory *)
	fbBuffer 	: FB_MemRingBuffer;(* Basic (lower level) buffer control function block *)
END_VAR

;

ACTION A_AddTail:
(* adds new fifo entry *)
fbBuffer.A_AddTail( 	pWrite:= ADR( putError ), cbWrite := SIZEOF( putError ),
					pBuffer:= ADR(buffer), cbBuffer:= SIZEOF(buffer),
					bOk=>bOk, nCount=>nCount );
IF bOk THEN
	IF bDbg THEN(* log message *)
		F_ADSLOGERROR( CONCAT( sDesc, '<=' ), putError );
	END_IF
END_IF
END_ACTION

ACTION A_RemoveHead:
(* removes oldest fifo entry *)
fbBuffer.A_RemoveHead( 	pRead := ADR(getError), cbRead := SIZEOF(getError),
						pBuffer:= ADR(buffer), cbBuffer:= SIZEOF(buffer),
						bOk=>bOk, nCount=>nCount );
END_ACTION

ACTION A_Reset:
(* resets fifo = clears all data *)
fbBuffer.A_Reset( pBuffer:= ADR(buffer), cbBuffer:= SIZEOF(buffer),
				bOk=>bOk, nCount=>nCount );
END_ACTION

END_FUNCTION_BLOCK

// ---- POUs/IP_POUs/F_ADSLOGERROR.TcPOU
FUNCTION F_ADSLOGERROR : DINT
(* This function logs communication error messages to the TwinCAT System Log View *)
VAR_INPUT
	sPrefix		: STRING(20);(* Debug message prefix string (allows the identification of log message source) *)
	nErrID		: DWORD; (* Error code *)
END_VAR

IF nErrId = 0 THEN
	F_ADSLOGERROR := ADSLOGSTR( ADSLOG_MSGTYPE_HINT OR ADSLOG_MSGTYPE_LOG, CONCAT( sPrefix, ' No error!   %s'),'' );
ELSIF (  nErrId AND DWORD#16#80000000 ) = 16#80000000 THEN
	F_ADSLOGERROR := ADSLOGDINT( ADSLOG_MSGTYPE_ERROR OR ADSLOG_MSGTYPE_LOG, CONCAT( sPrefix, ' Win32 error: %d' ), DWORD_TO_DINT(SCODE_CODE( nErrId )) );
ELSIF (nErrId AND 16#00008100) =16#00008100 THEN
	F_ADSLOGERROR := ADSLOGDINT( ADSLOG_MSGTYPE_ERROR OR ADSLOG_MSGTYPE_LOG, CONCAT( sPrefix, ' Internal PLC sample project (user) error: %d' ), DWORD_TO_DINT(nErrId) );
ELSIF (nErrId AND 16#00008000) =16#00008000 THEN
	F_ADSLOGERROR := ADSLOGDINT( ADSLOG_MSGTYPE_ERROR OR ADSLOG_MSGTYPE_LOG, CONCAT( sPrefix, ' Internal TCP/IP Connection Server error: %d' ), DWORD_TO_DINT(nErrId) );
ELSE
	F_ADSLOGERROR := ADSLOGDINT( ADSLOG_MSGTYPE_ERROR OR ADSLOG_MSGTYPE_LOG, CONCAT( sPrefix, ' TwinCAT System error: %d' ), DWORD_TO_DINT(nErrId) );
END_IF

END_FUNCTION

// ---- POUs/IP_POUs/SCODE_CODE.TcPOU
FUNCTION SCODE_CODE : DWORD
(* Helper function: returns the lower word of error code *)
VAR_INPUT
	sc		: DWORD;
END_VAR

SCODE_CODE := 16#FFFF AND sc;

END_FUNCTION

// ---- VISUs/HardStuff.TcVIS
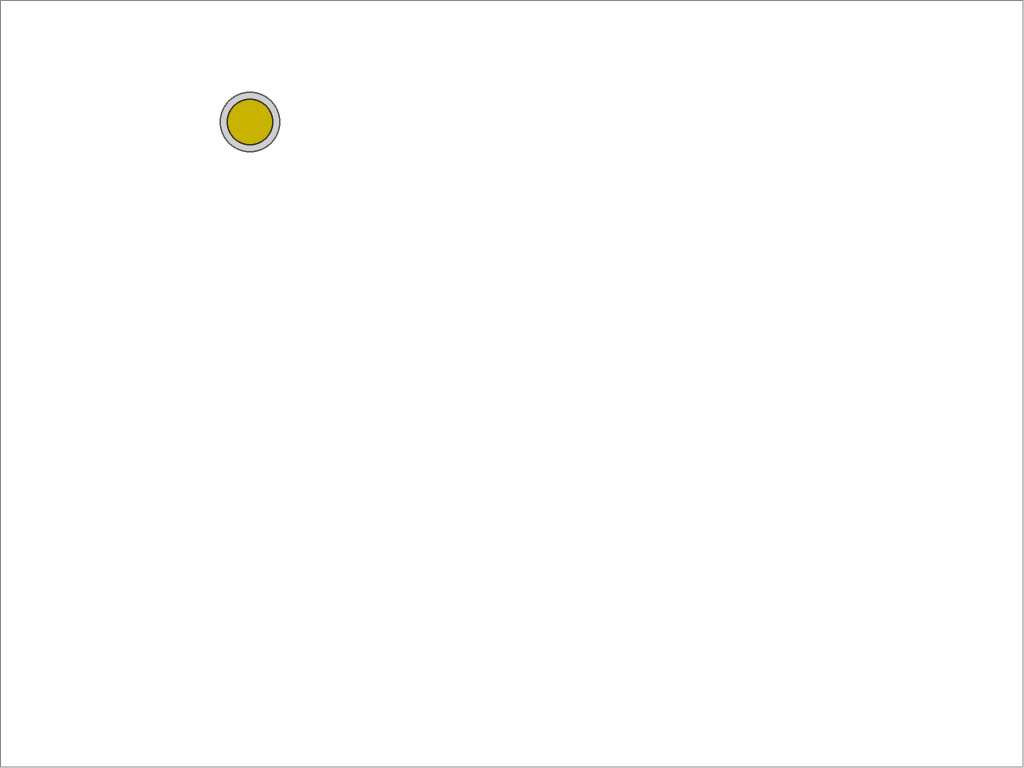
VISUALIZATION HardStuff  // 1024x768
    Lamp1 (215,87 70x70), style: Lamp-Lamp1-Yellow
END_VISUALIZATION
